PROGRAM P_EventHandling2
VAR
	sAktywnyEkran: STRING;
	i: INT;
	
	j: INT;
	k: INT;
	i2: INT;
	tonNieMaAlarmow: TON;
	bAlarm: BOOL;
	bOstrzezenie: BOOL;
	bAalrmLekki: BOOL;
END_VAR


//==============================================================
//		ukrywanie alarmów w stopce gdy otwarty ekran alarmów
IF GVL_HMI.hmiPanel.uiMenu=1 THEN
	
GVL_Event.bFilterActiveOnly2:=FALSE;
ELSE
	GVL_Event.bFilterActiveOnly2:=TRUE;
END_IF

//==============================================================
//     sprawdzenie czy jest alarm dla pokazania-ukrycia na stopce
//FOR i:=1 TO UDINT_TO_INT(GVL_EHS.diEventsDefinition) DO
FOR i:=1 TO 100 DO
	
	bAlarm:=GVL_EHS.arrEventDefinition[i].bActive;
	IF bAlarm THEN
		GVL_Event.bJestAalrm:=TRUE;
		EXIT;
		ELSE 
			GVL_Event.bJestAalrm:=FALSE;
		
	END_IF
	
END_FOR

FOR i2:=201 TO 300 DO
	
	bAalrmLekki:=GVL_EHS.arrEventDefinition[i2].bActive;
	IF bAalrmLekki THEN
		GVL_Event.bJestAalrmLekki:=TRUE;
		EXIT;
		ELSE 
			GVL_Event.bJestAalrmLekki:=FALSE;
	END_IF
END_FOR

FOR k:=101 TO 200 DO
	bOstrzezenie:=GVL_EHS.arrEventDefinition[k].bActive;
	IF bOstrzezenie THEN	
	GVL_Event.bJestOstrzezenie:=TRUE;
	EXIT;
		ELSE 
			GVL_Event.bJestOstrzezenie:=FALSE;
	END_IF
END_FOR
//===============================================================
//		ukrywanie alarmu na stopce
IF GVL_HMI.bResetAlarm THEN
	FOR j:=0 TO 200 DO
		GVL_Event.aAlarm[j]:=FALSE;
		GVL_Event.aWarning[j]:=FALSE;
	//	GVL_Event.aMessage[j]:=FALSE;
	END_FOR
	GVL_Event.bJestAalrm:=FALSE;
	GVL_Event.bJestAalrmLekki:=FALSE;
	GVL_Event.bJestOstrzezenie:=FALSE;
	//GVL_HMI.bResetAlarm:=FALSE;
END_IF

tonNieMaAlarmow(IN:=GVL_HMI.bResetAlarm , PT:=T#500MS , Q=> , ET=> );
IF tonNieMaAlarmow.Q THEN
	GVL_HMI.bResetAlarm:=FALSE;
END_IF

END_PROGRAM

(* stored: Version 1.1.0.1, ProductVersion 3.1.4024.15
   POU P_EventHandling2: Id {2812fc2b-4b1b-46f7-88e6-36a42cca0c43}, SpecialFunc None *)
